PROGRAM MAIN
VAR
	fbLog			: FB_Logger('MAIN');
	bWriteLog		: BOOL;
	bWriteCont		: BOOL;
	nVar1			: INT;
	nVar2			: T_MaxString;
	nVar3			: REAL;
END_VAR

VAR_TEMP
	fbContext		: FB_ContextBuilder;
END_VAR


IF bWriteLog OR bWriteCont THEN
	bWriteLog := FALSE;
	
	fbLog(
		eLogLevel	:= E_LogLEvel.eError,
		sMessage	:= 'Test Log Message {arg1} {arg2} {arg3}',
		stArg1		:= F_INT(nVar1),
		stArg2		:= F_String(nVar2),
		stArg3		:= F_REAL(nVar3),
		iContextBuilder := fbContext.WithContextInt('foo', 42).WithContextInt('bar', 420),
	);
	
	fbLog(
		eLogLevel	:= E_LogLEvel.eInfo,
		sMessage	:= 'Info Message',
	);

END_IF

Log4TC.CallLogTask();

END_PROGRAM

(* stored: Version 1.1.0.1, ProductVersion 3.1.4024.0
   POU MAIN: Id {9e023de9-a7d3-47c5-b36b-a81c12c72c93}, SpecialFunc None *)
